FUNCTION_BLOCK FB_SerialController
VAR_INPUT
	slaveNumber : INT;
END_VAR
VAR
	//fbEL6001	: FB_SerialCom;
	
	fbAsciiComm: FB_SerialCom;
	

	ReceiveStep: INT;
	ProcessVariableRead : BOOL;
	SetpointRead : BOOL;
	ProcessVariableReceived : BOOL;
	SetpointReceived : BOOL;
	SendStep: INT;
	bStartSend: BOOL;
	start3: BOOL;
	received3: BOOL;
	start4: BOOL;
	received4: BOOL;
	Setpoint: STRING;
	
	fbUpdateSetpoint: FB_UpdateSetpoint;
	pumpingPressureMeasurement: DINT;
	pumpingPressureSetpoint: DINT;
	pumpingPressureSetSetpoint: DINT;
	pumpingPressureSetSetpointPrev: DINT;
	tonMessageUpdate: TON;
	rTrigMessageNotUpdated: R_TRIG;
	OutputPowerRead: BOOL;
	OutputPowerReceived: BOOL;
	pumpingPressureOutputPower: DINT;
	testi: BOOL;
END_VAR

END_FUNCTION_BLOCK

(* stored: Version 1.1.0.1, ProductVersion 3.1.4024.9
   POU FB_SerialController: Id {d2970343-d39c-46df-9e3f-e9dac4aaac85}, SpecialFunc None *)
